TYPE ST_SensorData :
STRUCT
    SampleNumber    : INT;
    MeasurementNr   : INT;
    EncoderValue    : LREAL;
    Cap1Value       : LREAL;
    Cap2Value       : LREAL;
END_STRUCT
END_TYPE

(* stored: Version 1.1.0.1
   DUT ST_SensorData: Id {16fa3717-afac-47b4-939c-4d2e6d9441cb} *)
